(* CoDeSys 2.3.9.59 project: Nastro_Timer e Pulsante.pro *)
(* Libraries: STANDARD.LIB *)

(* Task configuration *)
TASK Standard (PRIORITY := 0, INTERVAL := T#10ms);
	MAIN
END_TASK

(* POU MAIN, LD *)
PROGRAM MAIN
VAR

	pezzo_magazzino  AT%IX0.0:BOOL;
	fine_corsa_nastro  AT%IX0.6:BOOL;
	pistone_avanti AT%IX0.2:BOOL;
	pistone_indietro AT%IX0.4:BOOL;
	pulsante:BOOL;

	nastro_on  AT%QX0.0:BOOL;
	pistone_on  AT%QX0.2:BOOL;
	bobina:BOOL;

	timer: TON;
	mytime: TIME;
END_VAR
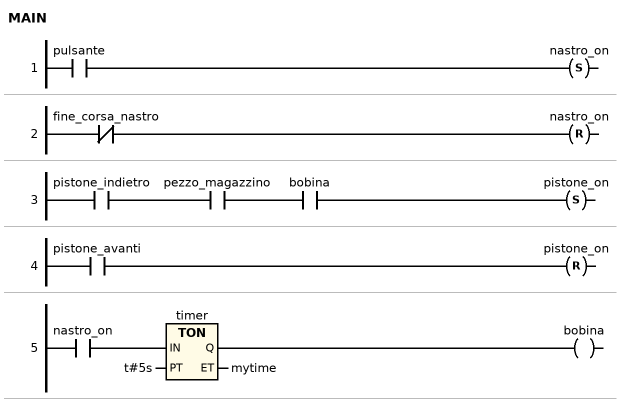
_LD_ (* Ladder Diagram *)
NETWORK 1
	[pulsante] --- (S nastro_on)
NETWORK 2
	[/fine_corsa_nastro] --- (R nastro_on)
NETWORK 3
	[pistone_indietro] - [pezzo_magazzino] - [bobina] --- (S pistone_on)
NETWORK 4
	[pistone_avanti] --- (R pistone_on)
NETWORK 5
	[nastro_on] - timer:TON(IN: *, PT: t#5s, ET => mytime) --- (bobina)
_END_LD_
(* the same logic as Structured Text *)
(* Network 1 *)
IF pulsante THEN nastro_on := TRUE; END_IF;
(* Network 2 *)
IF NOT fine_corsa_nastro THEN nastro_on := FALSE; END_IF;
(* Network 3 *)
IF pistone_indietro AND pezzo_magazzino AND bobina THEN pistone_on := TRUE; END_IF;
(* Network 4 *)
IF pistone_avanti THEN pistone_on := FALSE; END_IF;
(* Network 5 *)
timer(IN := nastro_on, PT := t#5s);
mytime := timer.ET;
bobina := timer.Q;
END_PROGRAM

(* Visualisation prova
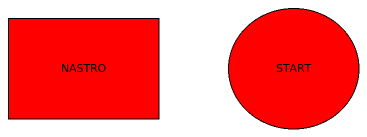
ellipse at (270,60)-(401,181): text "START"; toggles MAIN.nastro_on
rounded rectangle at (50,70)-(201,171): text "NASTRO"; alarm colour if MAIN.nastro_on
*)
